FUNCTION F_CheckAllOccupied : BOOL
(**************************************************************************************
 * 	Application		:	BoxControl Framework
 *	Revision		:	$Revision: 417092 $
 *	Revision date	:	$Date: 2018-11-14 12:58:58 +0100 (Mi., 14 Nov 2018) $
 *	Last changed by	:	$Author: q8aberh $
 *	URL				:	$URL: http://almscdc.swisslog.com/repo/SWPD/Development/ProMove/02_Controls/ProBox/03_Implementation/01_DevelopmentProject/01_Software/ProBox_COE/ProBox_DevProj_v1.0/PLC_1/20_Product/10_App/12_E_Functions/11_ProBox/02_Functions/02_TransportControl/F_Che $
 *
 *	Purpose			:	Return number of zones
 *
 * ------------------------------------------------------------------------------------
 *	Copyright Swisslog [IP AG], Switzerland. All rights reserved.
 * 
 * ------------------------------------------------------------------------------------
 *	
 * 	Revision History: 
 *
 * 	VERSION			DATE			INITIALS			DESCRIPTION
 *	0.1				01.01.2001		swl					Example
 *
 **************************************************************************************)
VAR_INPUT
	eFunctionNumber		: E_FunctionNumber; // Function number
END_VAR
VAR
	idx 				: INT; // Iterator
	AllOccupied			: BOOL; // Temp to check if all zones are free
END_VAR

// Check if function number is valid
IF eFunctionNumber > E_FunctionNumber.F_BEGIN_FUNCTION AND
   eFunctionNumber < E_FunctionNumber.F_END_FUNCTION THEN
  
   // Check reference is valid
   IF __ISVALIDREF(FunctionRegistry[eFunctionNumber].rSettingsFunction) THEN
		// Return All Occupied
		AllOccupied := TRUE;
		FOR idx := 1 TO FunctionRegistry[eFunctionNumber].rSettingsFunction.NumberOfZones DO
			IF NOT FunctionRegistry[eFunctionNumber].Zone[idx].refZoneData.TransportControlData.Occupied THEN
				AllOccupied := FALSE;
				EXIT;
			END_IF
		END_FOR
		F_CheckAllOccupied := AllOccupied;
   END_IF
END_IF

END_FUNCTION

(* stored: Version 1.1.0.1, ProductVersion 3.1.4024.4
   POU F_CheckAllOccupied: Id {0a365713-2c95-49ad-af8e-d0a3452744f4}, SpecialFunc None *)
